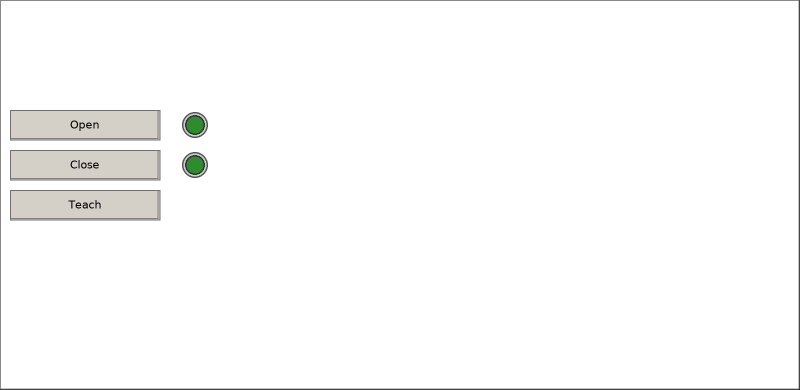
VISUALIZATION VisuValveControl  // 800x390
    Rectangle (0,0 800x390)
    Button (10,110 150x30), "Open"
        tap GVL_DevManual.fbManualControler.pDevValve^.stManualCtrl.bCmdOpen
    Button (10,150 150x30), "Close"
        tap GVL_DevManual.fbManualControler.pDevValve^.stManualCtrl.bCmdClose
    Lamp1 (180,110 30x30), variable: GVL_DevManual.fbManualControler.pDevValve^.bFco_Open, style: Lamp-Lamp1-Green
    Button (10,190 150x30), "Teach"
        toggle GVL_DevManual.fbManualControler.pDevValve^.stManualCtrl.bCmdTeach
    Lamp1 (180,150 30x30), variable: GVL_DevManual.fbManualControler.pDevValve^.bFco_Closed, style: Lamp-Lamp1-Green
END_VISUALIZATION

(* stored: Version 1.1.0.1, ProductVersion 3.1.4024.5
   Visu VisuValveControl: Id {5822c885-21b0-4bb6-89f5-b6fde4df3f46} *)
